// TIA Portal V19 export
TYPE "LAF_typeAxisDiagSensor"
TITLE = LAF_typeAxisDiagSensorStatus
// Status and actual values of an encoder of a Technology Object
// stored: Access Published
   STRUCT
      state { ExternalWritable := 'False'} : DInt;   // Status of actual encoder value (0=not valid, 1=waiting for valid status, 2=valid)
      communicationOK { ExternalWritable := 'False'} : Bool;   // Cyclic bus communication between controller and encoder / Cyclic bus communication between controller and encoder (FALSE = not established, TRUE = established)
      error { ExternalWritable := 'False'} : Bool;   // Error in the measuring system / FALSE = no error in the measuring system, TRUE = error in the measuring system
      control { ExternalWritable := 'False'} : Bool;   // Encoder is active / FALSE = encoder is not active, TRUE = encoder is active
      position { ExternalWritable := 'False'} : LReal;   // Encoder position
      velocity { ExternalWritable := 'False'} : LReal;   // Encoder velocity
      adaptionState { ExternalWritable := 'False'} : DInt;   // Status of automatic data transfer of encoder parameters (0=not adapted, 1=in adaption, 2=adapted, 3= not applicable, 4=adaption error)
      adjusted { ExternalWritable := 'False'} : DInt;   // Homing status of the encoder (0=not homed, 1=homed (with active homing, passive homing, absolute encoder adjustment, incremental encoder adjustment))
   END_STRUCT;
END_TYPE
